{attribute 'GeneratedUsingTerminal: EL6201-0000-0017'}
{attribute addProperty BoxType "EL6201-0000-0017"}
{attribute addProperty Id "Slave_21A_DO0BOOL1Slave_21A_DO1BOOL1Slave_21A_DO2BOOL1Slave_21A_DO3BOOL1Slave_21B_DO0BOOL1Slave_21B_DO1BOOL1Slave_21B_DO2BOOL1Slave_21B_DO3BOOL1"}
{attribute addProperty CRC "1247521479"}
{attribute addProperty Size "8"}
TYPE Slave_21_Outputs_4A5BAAC7 :
STRUCT
	{attribute addProperty Name "Slave_21A_DO0"}
	Slave_21A_DO0 : BOOL;
	{attribute addProperty Name "Slave_21A_DO1"}
	Slave_21A_DO1 : BOOL;
	{attribute addProperty Name "Slave_21A_DO2"}
	Slave_21A_DO2 : BOOL;
	{attribute addProperty Name "Slave_21A_DO3"}
	Slave_21A_DO3 : BOOL;
	{attribute addProperty Name "Slave_21B_DO0"}
	Slave_21B_DO0 : BOOL;
	{attribute addProperty Name "Slave_21B_DO1"}
	Slave_21B_DO1 : BOOL;
	{attribute addProperty Name "Slave_21B_DO2"}
	Slave_21B_DO2 : BOOL;
	{attribute addProperty Name "Slave_21B_DO3"}
	Slave_21B_DO3 : BOOL;
END_STRUCT
END_TYPE

(* stored: Version 1.2.0.0, ProductVersion 3.1.4024.9
   DUT Slave_21_Outputs_4A5BAAC7: Id {8f2ed994-2771-499c-8d34-4fb509946fce} *)
